// TIA Portal project "Comunicando_Socket" (V18)

(* hardware
DEVICE "ET 200SP station_1"  ET 200SP-Station
   slot 0: "Rack_0"  Rack  6ES5 710-8MAx1
   slot 1: "PLC_1"  CPU 1510SP-1 PN  6ES7 510-1DJ01-0AB0  V2.5
      slot 32768: "PROFINET interface_1"  X1
         slot 32771: "Port_3"  X1 P3
   slot 2: "Server module_1"  Server module  6ES7 193-6PA00-0AA0  V1.1
      slot 1: "Server module_1"  Server module
   slot 127: "BA 2xRJ45"  BA 2xRJ45  6ES7 193-6AR00-0AA0  V0.0
      slot 32769: "Port_1"  X1 P1  6ES7 193-6AR00-0AA0
      slot 32770: "Port_2"  X1 P2  6ES7 193-6AR00-0AA0
*)

// ===== PLC "PLC_1"  CPU 1510SP-1 PN =====

VAR_GLOBAL   // PLC tag table "Default tag table"
   "Clock_Byte" AT %MB0 : Byte;
   "Clock_10Hz" AT %M0.0 : Bool;
   "Clock_5Hz" AT %M0.1 : Bool;
   "Clock_2.5Hz" AT %M0.2 : Bool;
   "Clock_2Hz" AT %M0.3 : Bool;
   "Clock_1.25Hz" AT %M0.4 : Bool;
   "Clock_1Hz" AT %M0.5 : Bool;
   "Clock_0.625Hz" AT %M0.6 : Bool;
   "Clock_0.5Hz" AT %M0.7 : Bool;
END_VAR

DATA_BLOCK "TCON_params"   // DB5
{ S7_Optimized_Access := 'TRUE' }
VERSION : 0.1
   VAR
      Connection_Parameters : TCON_Param;
      Error : Bool;
      Busy : Bool;
      Status : Word;
      DONETCON : Bool;
      TCONSTART : Bool := true;
   END_VAR
BEGIN
   Connection_Parameters.ID := 1;
   Connection_Parameters.LOCAL_TSAP_ID[1] := 07;
   Connection_Parameters.LOCAL_TSAP_ID[2] := 229;
   Connection_Parameters.REM_STADDR[1] := 192;
   Connection_Parameters.REM_STADDR[2] := 168;
   Connection_Parameters.REM_STADDR[3] := 1;
   Connection_Parameters.REM_STADDR[4] := 123;
   Connection_Parameters.REM_TSAP_ID[1] := 7;
   Connection_Parameters.REM_TSAP_ID[2] := 228;
END_DATA_BLOCK

DATA_BLOCK "TCP_Data"   // DB6
{ S7_Optimized_Access := 'TRUE' }
VERSION : 0.1
   VAR
      Data_to_Send : DInt := 1234;
      Received_Array : Array[0..4] of Char;
      Sent_Array : Array[0..10] of Char;
      Received_Data : DInt;
   END_VAR
BEGIN
   Sent_Array[0] := 'H';
   Sent_Array[1] := 'E';
   Sent_Array[2] := 'L';
   Sent_Array[3] := 'L';
   Sent_Array[4] := 'O';
   Sent_Array[6] := 'W';
   Sent_Array[7] := 'O';
   Sent_Array[8] := 'R';
   Sent_Array[9] := 'L';
   Sent_Array[10] := 'D';
END_DATA_BLOCK

ORGANIZATION_BLOCK "Main"   // OB1, LAD, ProgramCycle
TITLE = "Main Program Sweep (Cycle)"
{ S7_Optimized_Access := 'TRUE' }
VERSION : 0.1
   VAR_INPUT
      Initial_Call : Bool;   // Initial call of this OB
      Remanence : Bool;   // =True, if remanent data are available
   END_VAR
BEGIN

REGION Network 1
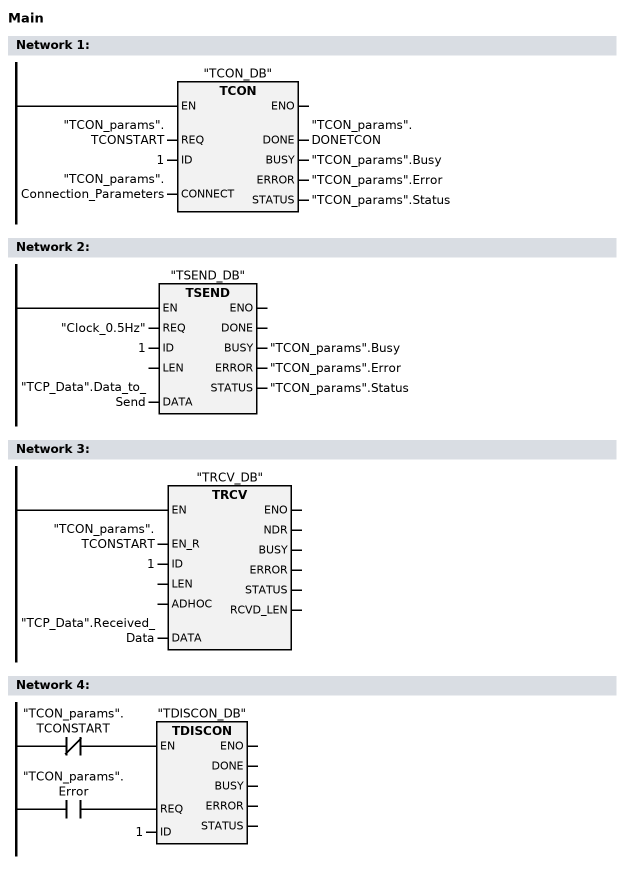
   "TCON_DB"(REQ := "TCON_params".TCONSTART,   // TCON
             ID := 1,
             CONNECT := "TCON_params".Connection_Parameters,
             DONE => "TCON_params".DONETCON,
             BUSY => "TCON_params".Busy,
             ERROR => "TCON_params".Error,
             STATUS => "TCON_params".Status);
END_REGION

REGION Network 2
   "TSEND_DB"(REQ := "Clock_0.5Hz",   // TSEND
              ID := 1,
              DATA := "TCP_Data".Data_to_Send,
              BUSY => "TCON_params".Busy,
              ERROR => "TCON_params".Error,
              STATUS => "TCON_params".Status);
END_REGION

REGION Network 3
   "TRCV_DB"(EN_R := "TCON_params".TCONSTART, ID := 1, DATA := "TCP_Data".Received_Data);   // TRCV
END_REGION

REGION Network 4
   IF NOT "TCON_params".TCONSTART THEN
       "TDISCON_DB"(REQ := "TCON_params".Error, ID := 1);   // TDISCON
   END_IF;
END_REGION
END_ORGANIZATION_BLOCK